# EPICS substitutions: nes_rte/nes_rteApp/Db/neslab_rte.substitutions
file neslab_rte.template { pattern
{ Sys	, Dev		, PORT		}
{ Depo	, "{Chill:1}"	, Depo_Chill1	}
}
